{attribute addProperty BoxType "EL6201-0000-0017"}
{attribute addProperty Id "Slave_6A_DO0BIT10.12541Slave_6A_DO1BIT10.12542Slave_6A_DO2BIT10.12543Slave_6A_DO3BIT10.12544Slave_6B_DO0BIT10.12545Slave_6B_DO1BIT10.12546Slave_6B_DO2BIT10.12547Slave_6B_DO3BIT10.12548"}
{attribute addProperty CRC "1447856911"}
{attribute addProperty SizeInBites "8"}
{attribute addProperty SizeInBytes "1"}
TYPE Slave_6_Outputs_564C8B0F :
STRUCT
	{attribute addProperty Name "Slave_6A_DO0"}
	Slave_6A_DO0 : BIT;
	{attribute addProperty Name "Slave_6A_DO1"}
	Slave_6A_DO1 : BIT;
	{attribute addProperty Name "Slave_6A_DO2"}
	Slave_6A_DO2 : BIT;
	{attribute addProperty Name "Slave_6A_DO3"}
	Slave_6A_DO3 : BIT;
	{attribute addProperty Name "Slave_6B_DO0"}
	Slave_6B_DO0 : BIT;
	{attribute addProperty Name "Slave_6B_DO1"}
	Slave_6B_DO1 : BIT;
	{attribute addProperty Name "Slave_6B_DO2"}
	Slave_6B_DO2 : BIT;
	{attribute addProperty Name "Slave_6B_DO3"}
	Slave_6B_DO3 : BIT;
END_STRUCT
END_TYPE

(* stored: Version 1.2.0.0, ProductVersion 3.1.4024.9
   DUT Slave_6_Outputs_564C8B0F: Id {2915001b-cd96-42fb-9a05-c527efda185d} *)
